// TIA Portal V17 export
// export: Created 2025-05-22T06:00:58.4284441Z, ExportSetting WithDefaults, DisplayName Totally Integrated Automation Portal, DisplayVersion V17 Update 8, DisplayName TIA Portal Openness, DisplayVersion V17 Update 8, DisplayName TIA Portal Version Control Interface, DisplayVersion V17, DisplayName SINAMICS Startdrive Advanced, DisplayVersion V17 SP2, DisplayName SINAMICS Startdrive G110M, G120, G120C, G120D, G120P, G115D, DisplayVersion V17 SP2, DisplayName SINAMICS Startdrive G130, G150, S120, S150, SINAMICS MV, S210, DisplayVersion V17 SP2, DisplayName STEP 7 Professional, DisplayVersion V17 Update 8, DisplayName SINUMERIK ONE STEP 7 Toolbox, DisplayVersion V17 Update 12, DisplayName SINUMERIK ONE PLC Basic Program Plus, DisplayVersion V17 Update 12, DisplayName SINUMERIK 840D sl STEP 7 Toolbox, DisplayVersion V17 Update 12, DisplayName STEP 7 Safety, DisplayVersion V17 Update 6, DisplayName WinCC Advanced, DisplayVersion V17 Update 8
DATA_BLOCK "DB7001_UNIT_1_MAIN_SAFETY_DOOR"   // DB7001
{ DB_Accessible_From_OPC_UA := 'FALSE' }
AUTHOR : ETXETAR
VERSION : 1.0
// stored: AutoNumber false, DBAccessibleFromOPCUA false, DBAccessibleFromWebserver true, InstanceOfName FB7001_SAFETY_DOOR, InstanceOfType FB
"FB7001_SAFETY_DOOR"
   // VAR_INPUT
   //    OPTIONS_0 : Byte;
   //    CLOSED_I : Bool;
   //    LOCKED_I : Bool;
   //    LOCK_CONDITIONS : Bool;
   //    UNLOCK_PARTIAL_CONDITIONS : Bool;
   //    HMI_REQ_LINE : Bool;
   //    PANEL_LOCK_UNLOCK_PUSHBUTTON : Bool;
   //    LOCK_AUTO_REQ : Bool;
   //    UNLOCK_AUTO_REQ : Bool;
   //    PNEUMATIC_DRIVE_UNBLOCKED : Bool;
   // END_VAR
   // VAR_OUTPUT
   //    NOT_CLOSED_AND_LOCKED_ALARM : Bool;
   //    PNEUMATIC_DRIVE_NOT_UNBLOCKED_ALARM : Bool;
   //    NOT_OPEN_ALARM : Bool;
   //    UNLOCK_REQUEST_SEOC_WRN : Bool;
   //    NOT_CLOSED_WRN : Bool;
   //    HMI_MOTION_EXECUTABILITY_LEFT : Bool;
   //    HMI_MOTION_EXECUTABILITY_RIGHT : Bool;
   //    HMI_MOTION_END_POS_LEFT : Bool;
   //    HMI_MOTION_END_POS_RIGHT : Bool;
   //    HMI_MOTION_ACTIVE_LEFT : Bool;
   //    HMI_MOTION_ACTIVE_RIGHT : Bool;
   //    UNLOCK : Bool;
   //    RED_LIGHT : Bool;
   //    GREEN_LIGHT : Bool;
   // END_VAR
   // VAR
   //    SAFETY_DOOR : "SAFETY_DOOR";
   // END_VAR
BEGIN
END_DATA_BLOCK
